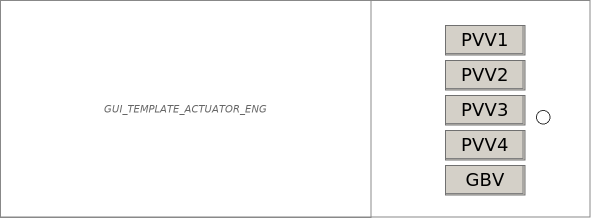
VISUALIZATION GUI_MICADO_Valves  // 591x218
    Frame (0,0 371x218)
        shows GUI_TEMPLATE_ACTUATOR_ENG(m_Cmd := MAIN.evac_micado.ptrVC[MAIN.evac_micado.guiValveIndex]^, m_Valve := MAIN.evac_micado.ptrV[MAIN.evac_micado.guiValveIndex]^)
    Button (445,25 80x30), "PVV1"
        OnMouseClick: execute { MAIN.evac_micado.guiValveIndex := 1; }
    Button (445,60 80x30), "PVV2"
        OnMouseClick: execute { MAIN.evac_micado.guiValveIndex := 2; }
    Button (445,95 80x30), "PVV3"
        OnMouseClick: execute { MAIN.evac_micado.guiValveIndex := 3; }
    Button (445,130 80x30), "PVV4"
        OnMouseClick: execute { MAIN.evac_micado.guiValveIndex := 4; }
    Button (445,165 80x30), "GBV"
        OnMouseClick: execute { MAIN.evac_micado.guiValveIndex := 5; }
    RadioButton (534,28 57x178), variable: MAIN.evac_micado.guiValveIndex-1
END_VISUALIZATION

(* stored: Version 1.1.0.1, ProductVersion 3.1.4024.9
   Visu GUI_MICADO_Valves: Id {e51f67e5-8e9b-46f1-8c41-db2a8d50e7ea} *)
